// TIA Portal project "Ofen" (V20)

(* hardware
DEVICE "S7-1500/ET200MP-Station_1"  S7-1500 station
   slot 0: "Profilschiene_0"  Rack  6ES7 590-1***0-0AA0
   slot 1: "PLC_1"  CPU 1513-1 PN  6ES7 513-1AM03-0AB0  V4.0
      slot 3: "CPU-Display_1"  6ES7591-1AA00-0AA0
      slot 32768: "PROFINET-Schnittstelle_1"  X1
         slot 32769: "Port_1"  X1 P1
         slot 32770: "Port_2"  X1 P2
      slot 34817: "Virtual CP interface port_1"  Virtual CP interface port  Virtual CP interface port FW V4.0
   slot 2: "DI 16x24VDC BA_1"  DI 16x24VDC BA  6ES7 521-1BH10-0AA0  V1.1
   slot 3: "DQ 16x24VDC/0.5A ST_1"  DQ 16x24VDC/0.5A ST  6ES7 522-1BH00-0AB0  V2.0
   slot 4: "AI 8xU/I/R/RTD BA_1"  AI 8xU/I/R/RTD BA  6ES7 531-7QF00-0AB0  V1.0
   slot 5: "AQ 8xU/I HS_1"  AQ 8xU/I HS  6ES7 532-5HF00-0AB0  V2.2
   slot 6: "AI 8xU/I HS_1"  AI 8xU/I HS  6ES7 531-7NF10-0AB0  V2.1
   slot 7: "AQ 8xU/I HS_2"  AQ 8xU/I HS  6ES7 532-5HF00-0AB0  V2.2
*)

// ===== PLC "PLC_1"  CPU 1513-1 PN =====

VAR_GLOBAL   // PLC tag table "Standard-Variablentabelle"
   "PlcLabConnectIn01" AT %ID32760 : DWord;
   "PlcLabConnectIn02" AT %ID32764 : DWord;
   "PlcLabConnectOut01" AT %QD32760 : DWord;
   "PlcLabConnectOut02" AT %QD32764 : DWord;
   "S1" AT %E0.0 : Bool;   // Betriebsschalter
   "M1" AT %A0.0 : Bool;   // Band_1
   "M2" AT %A0.1 : Bool;   // Band_2
   "M3" AT %A0.2 : Bool;   // Band_3
   "Gesamt_Temp" AT %MW36 : Int;   // Der Mittelwert von den drei Temperatursensoren.
   "H1" AT %A0.3 : Bool;   // Meldeleuchte für zu hohe Temperatur.
   "1b1_int" AT %MW30 : Int;   // Sensor 1 am Anfang des Ofens
   "1b2_int" AT %MW32 : Int;   // Sensor 2 in der Mitte des Ofens
   "1b3_int" AT %MW34 : Int;   // Sensor 3 am Ende des Ofens
   "D1" AT %AD30 : Real;   // Display zur Anzeige des Wertes
   "1b1" AT %ED30 : Real;
   "1b2" AT %ED34 : Real;
   "1b3" AT %ED38 : Real;
END_VAR

FUNCTION "Ofensteuerung" : Void   // FC1, FBD
{ S7_Optimized_Access := 'TRUE' }
VERSION : 0.1
   VAR_TEMP
      Temp1_konv : Real;
      Temp2_konv : Real;
      Temp3_konv : Real;
   END_VAR
   VAR CONSTANT
      Temp_zu_hoch : Int := 4000;   // Grenze für die Gesamttemperatur, die nicht höher als 400 Grad sein darf.
      Anzahl_Sensoren : Int := 3;
      Einheit_1 : Real := 10.0;   // Zum konvertieren in einen Kommawert fürs Display.
      Einheit_2 : Real := 3500.0;   // Zum konvertieren in Temperatur.
   END_VAR
BEGIN

REGION Network 1: Bandsteuerung
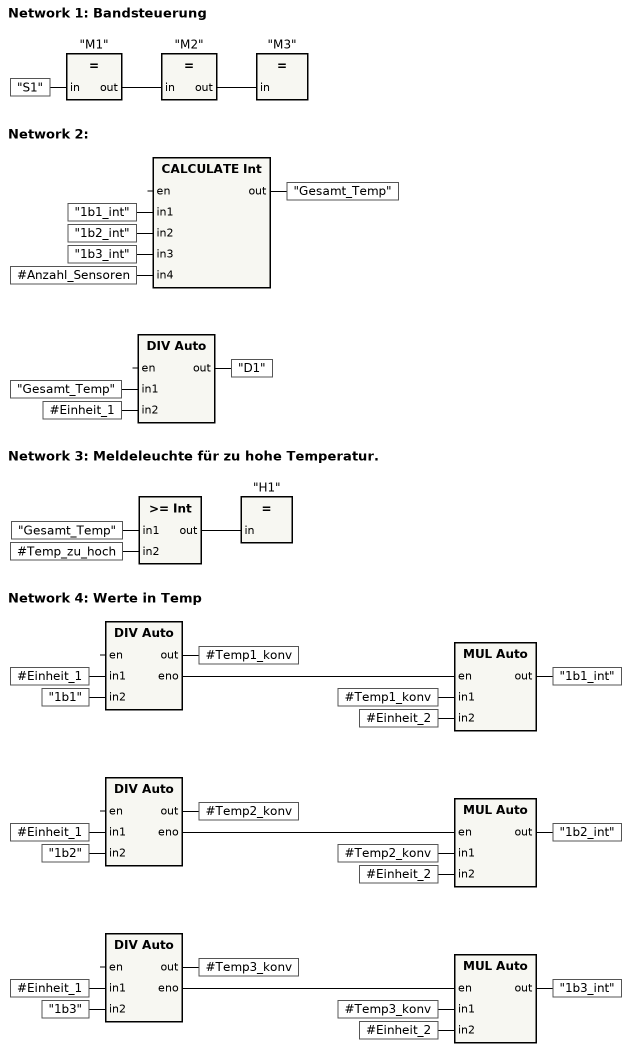
   "M1" := "S1";
   "M2" := "S1";
   "M3" := "S1";
END_REGION

REGION Network 2
   "Gesamt_Temp" := ("1b1_int"+"1b2_int"+"1b3_int")/#Anzahl_Sensoren;
   "D1" := "Gesamt_Temp" / #Einheit_1;
END_REGION

REGION Network 3: Meldeleuchte für zu hohe Temperatur.
   "H1" := "Gesamt_Temp" >= #Temp_zu_hoch;
END_REGION

REGION Network 4: Werte in Temp
   #Temp1_konv := #Einheit_1 / "1b1";
   "1b1_int" := #Temp1_konv * #Einheit_2;
   #Temp2_konv := #Einheit_1 / "1b2";
   "1b2_int" := #Temp2_konv * #Einheit_2;
   #Temp3_konv := #Einheit_1 / "1b3";
   "1b3_int" := #Temp3_konv * #Einheit_2;
END_REGION
END_FUNCTION

ORGANIZATION_BLOCK "Main"   // OB1, FBD, ProgramCycle
TITLE = "Main Program Sweep (Cycle)"
{ S7_Optimized_Access := 'TRUE' }
VERSION : 0.1
   VAR_INPUT
      Initial_Call : Bool;   // Initial call of this OB
      Remanence : Bool;   // =True, if remanent data are available
   END_VAR
BEGIN

REGION Network 1
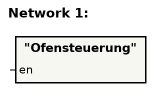
   "Ofensteuerung"();
END_REGION
END_ORGANIZATION_BLOCK